TYPE ST_MaterialContext :
STRUCT
	Id : STRING(80);
	OperationState : E_MaterialOperateState;
	// Add other information of wafer...
END_STRUCT
END_TYPE

(* stored: Version 1.1.0.1, ProductVersion 3.1.4026.18
   DUT ST_MaterialContext: Id {4b60fcdc-f719-468b-a244-a14310a360da} *)
